FUNCTION_BLOCK E_NOT
  (* Version 1.0, 2005-07-05, Goran Cengic, Chalmers *)
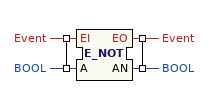
  EVENT_INPUT
    EI WITH A;
  END_EVENT
  EVENT_OUTPUT
    EO WITH AN;
  END_EVENT
  VAR_INPUT
    A : BOOL;
  END_VAR
  VAR_OUTPUT
    AN : BOOL := true;
  END_VAR
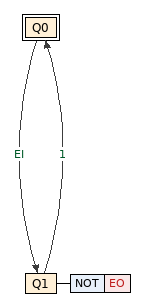
  EC_STATES
    Q0;
    Q1 : NOT -> EO;
  END_STATES
  EC_TRANSITIONS
    Q0 TO Q1 := EI;
    Q1 TO Q0 := 1;
  END_TRANSITIONS
  ALGORITHM NOT IN Java:
AN = !A;
  END_ALGORITHM
END_FUNCTION_BLOCK
